Yaskawa INFORM job: KRIS1A.JBI

/JOB
//NAME KRIS1A
//POS
///NPOS 195,195,193,7,0,0
///TOOL 0
///POSTYPE PULSE
///PULSE
C00000=15349,-87390,-111573,-674,86554,-86826
C00001=-110984,-87390,-111570,-673,86559,8331
C00002=-111759,-79535,-69021,-454,64406,8169
C00003=-114095,-78681,-67160,402,63698,7299
C00004=-114095,-78325,-65957,403,63140,7298
C00005=-114095,-78648,-67045,402,63644,7299
C00006=-113114,-93112,-73015,43,59884,7664
C00007=-114174,-91151,-70215,449,59172,7253
C00008=-114269,-89568,-69588,484,59599,7218
C00009=-112804,-96361,-75693,-76,59862,7786
C00010=-111133,-79411,-68712,-683,64284,8404
C00011=-110795,-77497,-66452,-807,63881,8532
C00012=-110795,-77213,-65470,-810,63423,8535
C00013=-111147,-78773,-67027,-680,63577,8402
C00014=-109795,-94038,-73387,-1221,59664,8950
C00015=-110034,-90449,-69592,-1136,59169,8863
C00016=-110197,-88771,-68919,-1070,59614,8797
C00017=-109724,-95740,-76085,-1239,60450,8969
C00018=-97790,-93891,-80845,-5517,64828,13352
C00019=-103428,-49774,-59623,-1029,84980,31565
C00020=-110091,-17957,-40687,2667,97599,44417
C00021=-110679,-18450,-38986,2708,96322,44197
C00022=-110679,-18552,-38259,2706,95822,44188
C00023=-109538,-18108,-38733,2608,96305,44575
C00024=-109458,-19366,-38871,2595,95741,44590
C00025=-109985,-19539,-38909,2643,95690,44414
C00026=-108888,-17833,-38981,2552,96578,44796
C00027=-113591,44136,17002,2949,94129,43179
C00028=-113558,44117,17472,2949,93828,43185
C00029=-113558,44084,18124,2949,93412,43175
C00030=-112698,44382,17754,2873,93761,43471
C00031=-112698,44348,18436,2870,93325,43460
C00032=-113010,44247,18329,2898,93349,43356
C00033=-112698,44452,16728,2876,94428,43485
C00034=-95102,58941,36484,-30043,98742,46310
C00035=-95139,59332,36927,-30037,98667,46316
C00036=-123036,27157,-10763,-19283,86742,21526
C00037=-150798,39984,8064,-10438,77055,13413
C00038=-150701,50951,18953,-20501,80603,7648
C00039=-146523,55066,28554,-32677,81611,-991
C00040=-149211,60857,35994,-32225,79233,-1370
C00041=-149211,60937,37447,-32305,78504,-1162
C00042=-149211,60857,35994,-32225,79233,-1370
C00043=-148938,63495,39015,-32331,78908,-1167
C00044=-149211,60857,35994,-32225,79233,-1370
C00045=-141139,35393,-539,-16647,85388,2500
C00046=-139001,60609,30102,-17411,80166,3961
C00047=-135441,52818,21854,-13680,80270,7361
C00048=-135777,54342,23766,-13597,79830,7293
C00049=-135777,54229,24881,-13624,79108,7374
C00050=-135777,54342,23766,-13597,79830,7293
C00051=-135623,56980,26711,-13659,79411,7392
C00052=-135777,54342,23766,-13597,79830,7293
C00053=-130150,67910,41047,-22097,81612,18545
C00054=-130308,68928,40049,-22014,82627,18301
C00055=-129747,65534,38183,-22158,82221,18578
C00056=-132405,65002,37751,-21584,81519,17750
C00057=-140354,55773,27245,-19636,81172,14970
C00058=-143966,58727,36324,-37580,82061,-623
C00059=-143233,57260,38729,-44506,80254,-83
C00060=-133755,47291,19718,-43086,89514,541
C00061=-130254,27624,-12420,-14523,95031,2735
C00062=-129705,29711,-12872,-15389,97022,78903
C00063=-131005,-814,-31676,-13890,80611,84029
C00064=-141281,-13707,-38556,3093,70993,82901
C00065=-136152,50678,21465,2134,66956,84718
C00066=-128094,56541,22144,-15053,77570,85372
C00067=-123724,-37006,-66316,-16306,84508,85949
C00068=-117270,-70326,-76879,-25476,75485,88799
C00069=-117396,-67861,-71382,-25671,73529,89185
C00070=-117796,-48019,-60604,-25175,76642,88348
C00071=-117668,-98678,-84753,-25780,65584,89666
C00072=-118323,-67765,-71239,-24397,72273,87906
C00073=-118030,-36635,-53581,-24971,77958,87975
C00074=-118346,-17679,-40448,-24750,79381,87560
C00075=-118238,-16726,-43675,-24636,81672,87118
C00076=-116459,-97013,-88147,-26591,69614,90459
C00077=-118030,-36635,-53581,-24971,77958,87975
C00078=-118346,-17679,-40448,-24750,79381,87560
C00079=-118238,-16726,-43675,-24636,81672,87118
C00080=-116459,-97013,-88147,-26591,69614,90459
C00081=-117668,-98678,-84753,-25780,65584,89666
C00082=-118323,-67765,-71239,-24397,72273,87906
C00083=-117271,-70296,-76864,-25474,75490,88797
C00084=-117270,-70326,-76879,-25476,75485,88799
C00085=-117396,-67861,-71382,-25671,73529,89185
C00086=-117796,-48019,-60604,-25175,76642,88348
C00087=-116979,-69120,-74771,-25636,74961,89025
C00088=-117994,-43372,-61454,-24127,91092,85341
C00089=-149498,-32155,-54450,-17063,84771,75512
C00090=-141330,-38704,-51094,-33432,76685,78426
C00091=-130528,-69811,-74379,-36386,79670,81887
C00092=-132947,-100822,-92962,-36380,74991,82451
C00093=15349,-87390,-111573,-674,86554,-86826
C00094=15349,-87390,-111573,-674,86554,-86826
C00095=15349,-87390,-111570,-674,86556,-86825
C00096=3643,-76224,-106676,19950,71810,76872
C00097=15349,-87390,-111570,-674,86556,-86825
C00098=-68824,-87390,-111568,-659,86557,2288
C00099=-102324,-63179,-76492,-4543,93838,9300
C00100=-99268,-62121,-71685,-4896,91607,10397
C00101=-101449,-61888,-70084,-4627,90618,9708
C00102=-101449,-61917,-69079,-4627,89987,9729
C00103=-101449,-61887,-70112,-4627,90636,9704
C00104=-98771,-79826,-78849,-4944,86964,10742
C00105=-97205,-87840,-78173,-7148,76765,11690
C00106=-97422,-86698,-77695,-7095,77039,11596
C00107=-98458,-92698,-83162,-6885,77230,11227
C00108=-70334,-47845,-62333,-11740,90555,19804
C00109=-68889,-44293,-58067,-11955,89977,20346
C00110=-68889,-44364,-57255,-11953,89453,20397
C00111=-68889,-44289,-58112,-11958,90008,20343
C00112=-63676,-56068,-65467,-12713,89294,22180
C00113=-64287,-54843,-62333,-12625,87932,22111
C00114=-64982,-53370,-61506,-12527,88068,21862
C00115=-63556,-56320,-65366,-12731,89128,22240
C00116=-105066,-71099,-78115,-5454,84680,8612
C00117=-111759,-50737,-67326,-4071,88105,-39576
C00118=-98977,-49335,-63615,-15063,89376,-36463
C00119=-99018,-49671,-62454,-15054,88511,-36372
C00120=-99018,-49749,-61553,-15054,87936,-36300
C00121=-99018,-49696,-62187,-15054,88340,-36350
C00122=-100915,-50718,-62779,-14728,87845,-36938
C00123=-100789,-50793,-62111,-14749,87431,-36845
C00124=-100259,-50517,-61951,-14840,87569,-36680
C00125=-101317,-50964,-63445,-14655,88049,-37098
C00126=-98850,-47982,-62812,-15085,89595,-36444
C00127=-99170,-48330,-61581,-15027,88634,-36434
C00128=-99170,-48394,-60912,-15027,88207,-36380
C00129=-99183,-48208,-61790,-15025,88819,-36461
C00130=-101244,-49312,-62437,-14669,88288,-37099
C00131=-100997,-49277,-61381,-14712,87718,-36948
C00132=-100426,-49069,-61280,-14811,87864,-36771
C00133=-101005,-49253,-62663,-14710,88495,-37043
C00134=-99461,-60085,-69932,-19764,73355,-34813
C00135=-111458,-11031,-30949,20838,73112,-726
C00136=-111844,18040,-3295,21202,74863,-1057
C00137=-111040,19701,-1743,20952,74565,-817
C00138=-111040,19683,-1004,20994,74127,-894
C00139=-110997,19721,-1737,20937,74560,-802
C00140=-111040,21506,-67,20957,74469,-835
C00141=-110997,19721,-1737,20937,74560,-802
C00142=-112260,2825,-16849,21290,75457,-1102
C00143=-114727,-25650,-50489,21683,81747,-843
C00144=-114727,-25650,-50489,21683,81747,-843
C00145=-78893,324,-30560,8500,76378,10543
C00146=-78852,391,-30517,8483,76382,10557
C00147=-79073,11131,-13779,8761,71676,10146
C00148=-79035,11094,-12929,8771,71138,10119
C00149=-79073,11131,-13779,8761,71676,10146
C00150=-79422,12797,-12298,8905,71656,10024
C00151=-79073,11131,-13779,8761,71676,10146
C00152=-90006,37360,13465,10198,74665,-440
C00153=-98018,29482,5428,6676,74813,1335
C00154=-100387,34080,10935,-7216,71995,-1662
C00155=-101325,39705,22013,-25009,65580,-3161
C00156=-101232,47576,34073,-36115,63714,-3272
C00157=-99101,24615,5399,-28066,67939,-3113
C00158=-101092,-2809,-21504,5594,61806,151
C00159=-116279,-103565,-87668,15153,52841,-6820
C00160=-136626,-108292,-100051,23905,62636,71559
C00161=-126647,-9226,-38971,10424,73423,75937
C00162=-126713,-9857,-28436,10885,66731,75311
C00163=-125013,58541,36859,10521,61560,75459
C00164=-125013,58363,29682,10151,65819,75847
C00165=-150812,-11611,-31149,38982,76943,71088
C00166=-150812,-11611,-31149,38982,76943,71088
C00167=-179059,-124163,-86099,46721,72567,55901
C00168=-188308,-108023,-75488,46296,78544,54278
C00169=-175675,-91816,-69705,45351,75449,58945
C00170=-166987,-75634,-62751,43730,73998,62467
C00171=-158229,-51102,-50131,41259,73376,66301
C00172=-153526,-28687,-35659,40655,73501,68565
C00173=-150180,-12513,-24053,39553,72873,69823
C00174=-150180,-12464,-30917,38869,76208,71082
C00175=-153640,-28797,-40554,40201,75834,69434
C00176=-153526,-28687,-35659,40655,73501,68565
C00177=-150180,-12513,-24053,39553,72873,69823
C00178=-153459,-29015,-37831,40437,74369,68941
C00179=-158928,-63138,-59452,42454,73735,66180
C00180=-166987,-75634,-62751,43730,73998,62467
C00181=-158229,-51102,-50131,41259,73376,66301
C00182=-167024,-76273,-64991,43548,74788,62799
C00183=-185238,-109581,-79609,46117,78191,55596
C00184=-188308,-108023,-75488,46296,78544,54278
C00185=-175675,-91816,-69705,45351,75449,58945
C00186=-181552,-118218,-82845,46514,74578,55658
C00187=-187474,-110161,-80368,46081,79459,55112
C00188=-145536,-97007,-88996,9555,84002,75248
C00189=-145251,-96121,-85437,9544,82257,75216
C00190=-99167,-97649,-86024,2499,78276,90872
C00191=-118631,-91766,-78858,25217,81137,84835
C00192=-117699,-93504,-86004,20553,84337,85672
C00193=-134531,-91540,-85241,22037,89209,80450
C00194=3161,-91504,-85468,2682,88050,79011
BC00000=115,663699,1075117
BC00001=171753,674879,306456
BC00002=55475,735323,199167
BC00003=55475,735323,199167
BC00004=55475,735323,199167
BC00005=55475,735323,199167
BC00006=55475,735323,199167
BC00007=55475,735323,199167
BC00008=55475,735323,199167
BC00009=55475,735323,199167
BC00010=108320,735323,199167
BC00011=108320,735323,199167
BC00012=108320,735323,199167
BC00013=108320,735323,199167
BC00014=108320,735323,199167
BC00015=108320,735323,199167
BC00016=108320,735323,199167
BC00017=108320,735323,199167
BC00018=108320,735323,199167
BC00019=108320,735323,199167
BC00020=108320,735323,199167
BC00021=108320,735323,199167
BC00022=108320,735323,199167
BC00023=108320,735323,199167
BC00024=108320,735323,199167
BC00025=108320,735323,199167
BC00026=108320,735323,199167
BC00027=108320,749563,199167
BC00028=108320,749563,199167
BC00029=108320,749563,199167
BC00030=108320,749563,199167
BC00031=108320,749563,199167
BC00032=108320,749563,199166
BC00033=108320,749563,199167
BC00034=108320,749563,199167
BC00035=108320,749563,199167
BC00036=153902,806828,124230
BC00037=190527,806828,124230
BC00038=190527,806828,124230
BC00039=190527,806828,124230
BC00040=190526,806828,124220
BC00041=190526,806828,124220
BC00042=190526,806828,124220
BC00043=190526,806828,124220
BC00044=190526,806828,124220
BC00045=190527,806828,124230
BC00046=190527,806828,124230
BC00047=170092,806828,124230
BC00048=170092,806828,124230
BC00049=170092,806828,124230
BC00050=170092,806828,124230
BC00051=170092,806828,124230
BC00052=170092,806828,124230
BC00053=170093,806828,124227
BC00054=170093,806828,124227
BC00055=170093,806828,124227
BC00056=170093,806828,124224
BC00057=170093,806828,124224
BC00058=170093,806828,124224
BC00059=170093,806828,124227
BC00060=170093,806828,124227
BC00061=170093,806828,124227
BC00062=170093,806828,124227
BC00063=170093,806828,124227
BC00064=170093,806828,124227
BC00065=170093,806828,124227
BC00066=170093,806828,124227
BC00067=170093,806828,124227
BC00068=170093,743154,124227
BC00069=170093,743154,124227
BC00070=170093,743154,124227
BC00071=170093,806828,124227
BC00072=170093,806828,124227
BC00073=170093,806828,124227
BC00074=170093,806828,124227
BC00075=170093,806828,124227
BC00076=170093,806828,124227
BC00077=170093,806828,124227
BC00078=170093,806828,124227
BC00079=170093,806828,124227
BC00080=170093,806828,124227
BC00081=170093,806828,124227
BC00082=170093,806828,124227
BC00083=170093,806828,124227
BC00084=170093,743154,124227
BC00085=170093,743154,124227
BC00086=170093,743154,124227
BC00087=170093,743154,124227
BC00088=170093,743154,124227
BC00089=170093,743154,124227
BC00090=170093,743154,124227
BC00091=170093,743154,124227
BC00092=170093,743154,124227
BC00093=115,663699,1075117
BC00094=115,663699,1075117
BC00095=115,663700,1075116
BC00096=199464,674570,1075173
BC00097=141263,687330,337717
BC00098=222435,751088,164876
BC00099=279925,751088,164876
BC00100=279925,751088,164876
BC00101=279925,751088,164876
BC00102=279925,751088,164876
BC00103=279925,751088,164876
BC00104=279925,751088,164876
BC00105=279925,751088,164876
BC00106=279925,751088,164876
BC00107=279925,751088,164876
BC00108=279925,751088,164876
BC00109=279925,751088,164876
BC00110=279925,751088,164876
BC00111=279925,751088,164876
BC00112=279925,751088,164876
BC00113=279925,751088,164876
BC00114=279925,751088,164876
BC00115=279925,751088,164876
BC00116=279925,751088,164876
BC00117=279925,751088,164876
BC00118=279925,751088,164876
BC00119=279925,751088,164876
BC00120=279925,751088,164876
BC00121=279925,751088,164876
BC00122=279925,751088,164876
BC00123=279925,751088,164876
BC00124=279925,751088,164876
BC00125=279925,751088,164876
BC00126=279925,839714,164876
BC00127=279925,839714,164876
BC00128=279925,839714,164876
BC00129=279925,839714,164876
BC00130=279925,839714,164876
BC00131=279925,839714,164876
BC00132=279925,839714,164876
BC00133=279925,839714,164876
BC00134=279925,839714,164876
BC00135=279925,839714,164876
BC00136=279925,834738,164876
BC00137=279925,834738,164876
BC00138=279925,834738,164876
BC00139=279925,834738,164876
BC00140=279925,834738,164876
BC00141=279925,834738,164876
BC00142=279925,834738,164876
BC00143=279925,834738,164876
BC00144=279925,762190,164876
BC00145=244896,762190,164876
BC00146=278481,826600,138122
BC00147=278481,826600,138122
BC00148=278481,826600,138122
BC00149=278481,826600,138122
BC00150=278481,826600,138122
BC00151=278481,826600,138122
BC00152=302666,794256,164873
BC00153=326440,794256,164873
BC00154=326440,794256,164873
BC00155=326440,794254,164874
BC00156=326440,794256,164873
BC00157=326440,794256,164873
BC00158=326440,794256,164873
BC00159=326440,794256,164873
BC00160=326440,794256,164873
BC00161=326440,794256,164873
BC00162=326885,794948,164297
BC00163=326885,794948,164297
BC00164=326885,794948,164297
BC00165=326885,794948,164297
BC00166=326885,794948,164297
BC00167=326885,794948,164297
BC00168=326885,794948,164297
BC00169=326885,794948,164297
BC00170=326885,794948,164297
BC00171=326885,794948,164297
BC00172=326885,794948,164297
BC00173=326885,794948,164297
BC00174=326885,794948,164297
BC00175=326885,794948,164297
BC00176=326885,794948,164297
BC00177=326885,794948,164297
BC00178=326885,794948,164297
BC00179=326885,794948,164297
BC00180=326885,794948,164297
BC00181=326885,794948,164297
BC00182=326885,794948,164297
BC00183=326885,794948,164297
BC00184=326885,794948,164297
BC00185=326885,794948,164297
BC00186=326885,794948,164297
BC00187=326885,794948,164297
BC00188=326885,794948,164297
BC00189=326885,794948,164297
BC00190=326885,794948,164297
BC00191=326885,794948,164295
BC00192=326885,794948,164295
BC00193=326885,737668,213736
BC00194=87842,675035,1040975
EC00000=798157,0
EC00001=798154,2
EC00002=798154,2
EC00003=798154,2
EC00004=798154,2
EC00005=798154,2
EC00006=798154,2
EC00007=798154,2
EC00008=798154,2
EC00009=798154,2
EC00010=798154,2
EC00011=798154,2
EC00012=798154,2
EC00013=798154,2
EC00014=798154,2
EC00015=798154,2
EC00016=798154,2
EC00017=798154,2
EC00018=798154,2
EC00019=798154,2
EC00020=798154,2
EC00021=798154,2
EC00022=798154,2
EC00023=798154,2
EC00024=798154,2
EC00025=798154,2
EC00026=798154,2
EC00027=798154,2
EC00028=798154,2
EC00029=798154,2
EC00030=798154,2
EC00031=798154,2
EC00032=798153,2
EC00033=798154,2
EC00034=798154,2
EC00035=798154,2
EC00036=798154,2
EC00037=798154,2
EC00038=798154,2
EC00039=798154,2
EC00040=798150,3
EC00041=798150,3
EC00042=798150,3
EC00043=798150,3
EC00044=798150,3
EC00045=798154,2
EC00046=798154,2
EC00047=798154,2
EC00048=798154,2
EC00049=798154,2
EC00050=798154,2
EC00051=798154,2
EC00052=798154,2
EC00053=798153,2
EC00054=798151,3
EC00055=798151,3
EC00056=798152,2
EC00057=798153,2
EC00058=798153,2
EC00059=798153,2
EC00060=798153,2
EC00061=798153,2
EC00062=798153,2
EC00063=798153,2
EC00064=798153,2
EC00065=798153,2
EC00066=798153,2
EC00067=798153,2
EC00068=798153,2
EC00069=798153,2
EC00070=798153,2
EC00071=798153,2
EC00072=798153,2
EC00073=798153,2
EC00074=798153,2
EC00075=798153,2
EC00076=798153,2
EC00077=798153,2
EC00078=798153,2
EC00079=798153,2
EC00080=798153,2
EC00081=798153,2
EC00082=798153,2
EC00083=798153,2
EC00084=798153,2
EC00085=798153,2
EC00086=798153,2
EC00087=798153,2
EC00088=798153,2
EC00089=798153,2
EC00090=798153,2
EC00091=798157,0
EC00092=93266,10480
EC00093=184298,1105644
EC00094=798157,1112952
EC00095=798157,1112952
EC00096=798156,1112951
EC00097=798156,1112951
EC00098=798156,1112951
EC00099=798156,1112951
EC00100=798156,1112951
EC00101=798156,1112951
EC00102=798156,1112951
EC00103=798156,1112951
EC00104=798156,1112951
EC00105=798156,1112951
EC00106=798156,1112951
EC00107=798156,1112951
EC00108=798156,1112951
EC00109=798156,1112951
EC00110=798156,1112951
EC00111=798156,1112951
EC00112=798156,1112951
EC00113=798156,1112951
EC00114=798156,1112951
EC00115=798156,1112951
EC00116=798156,1112951
EC00117=798156,1112951
EC00118=798156,1112951
EC00119=798156,1112951
EC00120=798156,1112951
EC00121=798156,1112951
EC00122=798156,1112951
EC00123=798156,1112951
EC00124=798156,1112951
EC00125=798156,1112951
EC00126=798156,1112951
EC00127=798156,1112951
EC00128=798156,1112951
EC00129=798156,1112951
EC00130=798156,1112951
EC00131=798156,1112951
EC00132=798156,1112951
EC00133=798156,1112951
EC00134=798156,1112951
EC00135=798156,1112951
EC00136=798156,1112951
EC00137=798156,1112951
EC00138=798156,1112951
EC00139=798156,1112951
EC00140=798156,1112951
EC00141=798156,1112951
EC00142=798156,1112951
EC00143=798156,1112951
EC00144=798156,1112951
EC00145=798156,1112951
EC00146=798156,1112951
EC00147=798156,1112951
EC00148=798156,1112951
EC00149=798156,1112951
EC00150=798155,1112950
EC00151=798155,1112950
EC00152=798155,1112950
EC00153=798155,1112950
EC00154=798155,1112950
EC00155=798155,1112950
EC00156=798155,1112950
EC00157=798155,1112950
EC00158=798155,1112950
EC00159=798155,1112950
EC00160=798155,1112950
EC00161=798155,1112950
EC00162=798155,1112950
EC00163=798155,1112950
EC00164=798155,1112950
EC00165=798155,1112950
EC00166=798155,1112950
EC00167=798155,1112950
EC00168=798155,1112950
EC00169=798155,1112950
EC00170=798155,1112950
EC00171=798155,1112950
EC00172=798155,1112950
EC00173=798155,1112950
EC00174=798155,1112950
EC00175=798155,1112950
EC00176=798155,1112950
EC00177=798155,1112950
EC00178=798155,1112950
EC00179=798155,1112950
EC00180=798155,1112950
EC00181=798155,1112950
EC00182=798155,1112950
EC00183=798155,1112950
EC00184=798155,1112950
EC00185=798155,1112950
EC00186=798155,1112950
EC00187=798155,1112950
EC00188=798155,1112950
EC00189=798154,1112948
EC00190=798154,1112948
EC00191=798154,1112948
EC00192=798154,1103372
///POSTYPE BASE
///RECTAN
///RCONF 0,0,0,0,0,0,0,0,0,0,0,0,0,0,0,0,0,0,0,0,0,0,0,0
P00006=0.222,-3.123,-1.508,0.0000,0.0000,0.0000
P00021=-0.225,-6.128,-0.405,0.0000,0.0000,0.0000
P00022=0.222,-3.123,-1.508,0.0000,0.0000,0.0000
P00023=0.143,-0.036,0.682,0.0000,0.0000,0.0000
P00024=0.145,-0.552,1.326,0.0000,0.0000,0.0000
P00025=-2.003,0.006,0.728,0.0000,0.0000,0.0000
P00026=0.562,-0.002,-0.337,0.0000,0.0000,0.0000
//INST
///DATE 2025/03/14 13:10
///ATTR SC,RW
///GROUP1 RB1,BS1
///GROUP2 ST1
NOP
CALL JOB:CLEAN-R1_KM_3P
MOVJ C00000 BC00000 VJ=100.00  +MOVJ EC00000 VJ=100.00
MOVJ C00001 BC00001 VJ=100.00  +MOVJ EC00001 VJ=100.00
MOVJ C00002 BC00002 VJ=100.00  +MOVJ EC00002 VJ=100.00
SMOVL C00003 BC00003 V=100.0  +MOVJ EC00003
SREFP 3 C00004 BC00004  +REFP EC00004
CALL JOB:SEARCH-R1-S13D
SET P023 P006
SFTON3D P023
SMOVL C00005 BC00005 V=133.3  +MOVJ EC00005
SMOVL C00006 BC00006 V=133.3  +MOVJ EC00006
SMOVL C00007 BC00007 V=133.3  +MOVJ EC00007
SREFP 3 C00008 BC00008  +REFP EC00008
CALL JOB:SEARCH-R1-S13D
SET P023 P006
SFTON3D P023
SMOVL C00009 BC00009 V=166.7  +MOVJ EC00009
SFTOF3D
SMOVL C00010 BC00010 V=250.0  +MOVJ EC00010
SMOVL C00011 BC00011 V=100.0  +MOVJ EC00011
SREFP 3 C00012 BC00012  +REFP EC00012
CALL JOB:SEARCH-R1-S13D
SET P024 P006
SFTON3D P024
SMOVL C00013 BC00013 V=133.3  +MOVJ EC00013
SMOVL C00014 BC00014 V=133.3  +MOVJ EC00014
SMOVL C00015 BC00015 V=133.3  +MOVJ EC00015
SREFP 3 C00016 BC00016  +REFP EC00016
CALL JOB:SEARCH-R1-S13D
SET P024 P006
SFTON3D P024
SMOVL C00017 BC00017 V=166.7  +MOVJ EC00017
SFTOF3D
MOVJ C00018 BC00018 VJ=100.00  +MOVJ EC00018 VJ=100.00
MOVJ C00019 BC00019 VJ=100.00  +MOVJ EC00019 VJ=100.00
MOVJ C00020 BC00020 VJ=100.00  +MOVJ EC00020 VJ=100.00
SMOVL C00021 BC00021 V=100.0  +MOVJ EC00021
SREFP 3 C00022 BC00022  +REFP EC00022
CALL JOB:SEARCH-R1-S13D
SET P025 P006
SFTON3D P025
SMOVL C00023 BC00023 V=100.0  +MOVJ EC00023
SMOVL C00024 BC00024 V=100.0  +MOVJ EC00024
SREFP 3 C00025 BC00025  +REFP EC00025
CALL JOB:SEARCH-R1-S13D
SET P025 P006
SFTON3D P025
SMOVL C00026 BC00026 V=100.0  +MOVJ EC00026
SFTOF3D
SMOVL C00027 BC00027 V=500.0  +MOVJ EC00027
SMOVL C00028 BC00028 V=100.0  +MOVJ EC00028
SREFP 3 C00029 BC00029  +REFP EC00029
CALL JOB:SEARCH-R1-S13D
SET P026 P006
SFTON3D P026
SMOVL C00030 BC00030 V=133.3  +MOVJ EC00030
SMOVL C00031 BC00031 V=100.0  +MOVJ EC00031
SREFP 3 C00032 BC00032  +REFP EC00032
CALL JOB:SEARCH-R1-S13D
SET P026 P006
SFTON3D P026
SMOVL C00033 BC00033 V=166.7  +MOVJ EC00033
SFTOF3D
SMOVL C00034 BC00034 V=500.0  +MOVJ EC00034
MOVJ C00035 BC00035 VJ=100.00  +MOVJ EC00035 VJ=100.00
MOVJ C00036 BC00036 VJ=100.00  +MOVJ EC00036 VJ=20.00
MOVJ C00037 BC00037 VJ=20.00  +MOVJ EC00037 VJ=20.00
MOVJ C00038 BC00038 VJ=20.00  +MOVJ EC00038 VJ=20.00
MOVJ C00039 BC00039 VJ=20.00  +MOVJ EC00039 VJ=20.00
SMOVL C00040 BC00040 V=100.0  +MOVJ EC00040
SREFP 3 C00041 BC00041  +REFP EC00041
CALL JOB:SEARCH-R1-S13D
SET P022 P006
SFTON3D P022
SMOVL C00042 BC00042 V=100.0  +MOVJ EC00042
SREFP 3 C00043 BC00043  +REFP EC00043
CALL JOB:SEARCH-R1-S13D
SET P022 P006
SFTON3D P022
SMOVL C00044 BC00044 V=100.0  +MOVJ EC00044
SFTOF3D
MOVL C00045 BC00045 V=500.0  +MOVJ EC00045 VJ=20.00
MOVL C00046 BC00046 V=500.0  +MOVJ EC00046 VJ=20.00
SMOVL C00047 BC00047 V=500.0  +MOVJ EC00047
SMOVL C00048 BC00048 V=100.0  +MOVJ EC00048
SREFP 3 C00049 BC00049  +REFP EC00049
CALL JOB:SEARCH-R1-S13D
SET P021 P006
SFTON3D P021
SMOVL C00050 BC00050 V=100.0  +MOVJ EC00050
SREFP 3 C00051 BC00051  +REFP EC00051
CALL JOB:SEARCH-R1-S13D
SET P021 P006
SFTON3D P021
SMOVL C00052 BC00052 V=100.0  +MOVJ EC00052
MACRO1 MJ#(0) ARGF21
SMOVL C00053 BC00053 V=250.0  +MOVJ EC00053
REFP 1 RB1 C00054 BC00054
REFP 2 RB1 C00055 BC00055
ARCON
SWVON WEV#(100)
SMOVL C00056 BC00056 V=8.3  +MOVJ EC00054
SFTON3D P022
SMOVL C00057 BC00057 V=8.3  +MOVJ EC00055
SMOVL C00058 BC00058 V=8.3  +MOVJ EC00056
SMOVL C00059 BC00059 V=8.3  +MOVJ EC00057
ARCOF
SWVOF
SFTOF3D
SMOVL C00060 BC00060 V=333.3  +MOVJ EC00058
SMOVL C00061 BC00061 V=666.7  +MOVJ EC00059
MOVJ C00062 BC00062 VJ=100.00  +MOVJ EC00060 VJ=20.00
MOVJ C00063 BC00063 VJ=70.00  +MOVJ EC00061 VJ=20.00
MACRO1 MJ#(0) ARGF20
SFTON3D P025
SMOVL C00064 BC00064 V=250.0  +MOVJ EC00062
ARCON
SFTON3D P026
SMOVL C00065 BC00065 V=7.5  +MOVJ EC00063
ARCOF
SWVOF
SFTOF3D
SMOVL C00066 BC00066 V=333.3  +MOVJ EC00064
SMOVL C00067 BC00067 V=666.7  +MOVJ EC00065
SFTOF3D
MACRO1 MJ#(0) ARGF14
SMOVL C00068 BC00068 V=500.0  +MOVJ EC00066
SFTON3D P025
SMOVL C00069 BC00069 V=166.7  +MOVJ EC00067
ARCON
SWVON WEV#(20)
SMOVL C00070 BC00070 V=10.0  +MOVJ EC00068
SFTON3D P025
SMOVL C00071 BC00071 V=10.0  +MOVJ EC00069
SFTON3D P026
SMOVL C00072 BC00072 V=10.0  +MOVJ EC00070
SFTON3D P026
SMOVL C00073 BC00073 V=10.0  +MOVJ EC00071
SMOVL C00074 BC00074 V=10.0  +MOVJ EC00072
ARCOF
SWVOF
SMOVL C00075 BC00075 V=250.0  +MOVJ EC00073
SMOVL C00076 BC00076 V=500.0  +MOVJ EC00074
COMM MACRO1 MJ#(0) ARGF14
COMM SFTON3D P026
COMM SMOVL C00077 BC00077 V=250.0  +MOVJ EC00075
COMM ARCON
COMM SWVON WEV#(20)
COMM SMOVL C00078 BC00078 V=10.0  +MOVJ EC00076
COMM ARCOF
COMM SWVOF
COMM SMOVL C00079 BC00079 V=250.0  +MOVJ EC00077
COMM SMOVL C00080 BC00080 V=500.0  +MOVJ EC00078
COMM SFTON3D P025
COMM SMOVL C00081 BC00081 V=166.7  +MOVJ EC00079
COMM ARCON
COMM SWVON WEV#(20)
COMM SFTON3D P026
COMM SMOVL C00082 BC00082 V=9.2  +MOVJ EC00080
COMM ARCOF
COMM SWVOF
COMM SMOVL C00083 BC00083 V=250.0  +MOVJ EC00081
COMM SFTOF3D
COMM SMOVL C00084 BC00084 V=500.0  +MOVJ EC00082
COMM SFTON3D P025
COMM SMOVL C00085 BC00085 V=166.7  +MOVJ EC00083
COMM ARCON
COMM SWVON WEV#(20)
COMM SMOVL C00086 BC00086 V=10.0  +MOVJ EC00084
COMM ARCOF
COMM SWVOF
SFTOF3D
SMOVL C00087 BC00087 V=333.3  +MOVJ EC00085
SFTON3D P024
SMOVL C00088 BC00088 V=166.7  +MOVJ EC00086
ARCON
SWVON WEV#(20)
SFTON3D P023
SMOVL C00089 BC00089 V=12.5  +MOVJ EC00087
SMOVL C00090 BC00090 V=12.5  +MOVJ EC00088
ARCOF
SWVOF
SFTOF3D
SMOVL C00091 BC00091 V=500.0  +MOVJ EC00089
SMOVL C00092 BC00092 V=1000.0  +MOVJ EC00090
MOVJ C00093 BC00093 VJ=100.00  +MOVJ EC00091 VJ=20.00
MOVJ C00094 BC00094 VJ=100.00  +MOVJ EC00092 VJ=100.00
MOVJ C00095 BC00095 VJ=100.00  +MOVJ EC00093 VJ=100.00
MOVJ C00096 BC00096 VJ=100.00  +MOVJ EC00094 VJ=100.00
'DRUGA STRONA
CALL JOB:CLEAN-R1_KM_NEW
MOVJ C00097 BC00097 VJ=100.00  +MOVJ EC00095 VJ=100.00
MOVJ C00098 BC00098 VJ=100.00  +MOVJ EC00096 VJ=100.00
MOVJ C00099 BC00099 VJ=100.00  +MOVJ EC00097 VJ=100.00
MOVJ C00100 BC00100 VJ=100.00  +MOVJ EC00098 VJ=100.00
SMOVL C00101 BC00101 V=166.7  +MOVJ EC00099
SREFP 3 C00102 BC00102  +REFP EC00100
CALL JOB:SEARCH-R1-S13D
SET P023 P006
SFTON3D P023
SMOVL C00103 BC00103 V=250.0  +MOVJ EC00101
SMOVL C00104 BC00104 V=250.0  +MOVJ EC00102
SMOVL C00105 BC00105 V=250.0  +MOVJ EC00103
SREFP 3 C00106 BC00106  +REFP EC00104
CALL JOB:SEARCH-R1-S13D
SET P023 P006
SFTON3D P023
SFTOF3D
SMOVL C00107 BC00107 V=250.0  +MOVJ EC00105
SMOVL C00108 BC00108 V=250.0  +MOVJ EC00106
SMOVL C00109 BC00109 V=250.0  +MOVJ EC00107
SREFP 3 C00110 BC00110  +REFP EC00108
CALL JOB:SEARCH-R1-S13D
SET P024 P006
SFTON3D P024
SMOVL C00111 BC00111 V=250.0  +MOVJ EC00109
SMOVL C00112 BC00112 V=250.0  +MOVJ EC00110
SMOVL C00113 BC00113 V=250.0  +MOVJ EC00111
SREFP 3 C00114 BC00114  +REFP EC00112
CALL JOB:SEARCH-R1-S13D
SET P024 P006
SFTON3D P024
SFTOF3D
SMOVL C00115 BC00115 V=250.0  +MOVJ EC00113
MOVJ C00116 BC00116 VJ=100.00  +MOVJ EC00114 VJ=100.00
MOVJ C00117 BC00117 VJ=100.00  +MOVJ EC00115 VJ=100.00
MOVJ C00118 BC00118 VJ=100.00  +MOVJ EC00116 VJ=100.00
SMOVL C00119 BC00119 V=250.0  +MOVJ EC00117
SREFP 3 C00120 BC00120  +REFP EC00118
CALL JOB:SEARCH-R1-S13D
SET P025 P006
SFTON3D P025
SMOVL C00121 BC00121 V=250.0  +MOVJ EC00119
SMOVL C00122 BC00122 V=250.0  +MOVJ EC00120
SMOVL C00123 BC00123 V=100.0  +MOVJ EC00121
SREFP 3 C00124 BC00124  +REFP EC00122
CALL JOB:SEARCH-R1-S13D
SET P025 P006
SFTON3D P025
SFTOF3D
SMOVL C00125 BC00125 V=100.0  +MOVJ EC00123
SMOVL C00126 BC00126 V=333.3  +MOVJ EC00124
SMOVL C00127 BC00127 V=250.0  +MOVJ EC00125
SREFP 3 C00128 BC00128  +REFP EC00126
CALL JOB:SEARCH-R1-S13D
SET P026 P006
SFTON3D P026
SMOVL C00129 BC00129 V=250.0  +MOVJ EC00127
SMOVL C00130 BC00130 V=250.0  +MOVJ EC00128
SMOVL C00131 BC00131 V=100.0  +MOVJ EC00129
SREFP 3 C00132 BC00132  +REFP EC00130
CALL JOB:SEARCH-R1-S13D
SET P026 P006
SFTON3D P026
SFTOF3D
SMOVL C00133 BC00133 V=250.0  +MOVJ EC00131
SMOVL C00134 BC00134 V=333.3  +MOVJ EC00132
MOVJ C00135 BC00135 VJ=20.00  +MOVJ EC00133 VJ=20.00
MOVJ C00136 BC00136 VJ=20.00  +MOVJ EC00134 VJ=20.00
SMOVL C00137 BC00137 V=250.0  +MOVJ EC00135
SREFP 3 C00138 BC00138  +REFP EC00136
CALL JOB:SEARCH-R1-S13D
SET P021 P006
SFTON3D P021
SMOVL C00139 BC00139 V=250.0  +MOVJ EC00137
SREFP 3 C00140 BC00140  +REFP EC00138
CALL JOB:SEARCH-R1-S13D
SET P021 P006
SFTON3D P021
SFTOF3D
SMOVL C00141 BC00141 V=250.0  +MOVJ EC00139
MOVL C00142 BC00142 V=250.0  +MOVJ EC00140 VJ=20.00
MOVL C00143 BC00143 V=333.3  +MOVJ EC00141 VJ=20.00
SMOVL C00144 BC00144 V=1000.0  +MOVJ EC00142
SMOVL C00145 BC00145 V=1000.0  +MOVJ EC00143
SMOVL C00146 BC00146 V=250.0  +MOVJ EC00144
SMOVL C00147 BC00147 V=250.0  +MOVJ EC00145
SREFP 3 C00148 BC00148  +REFP EC00146
CALL JOB:SEARCH-R1-S13D
SET P022 P006
SFTON3D P022
SMOVL C00149 BC00149 V=250.0  +MOVJ EC00147
SREFP 3 C00150 BC00150  +REFP EC00148
CALL JOB:SEARCH-R1-S13D
SET P022 P006
SFTON3D P022
SFTOF3D
SMOVL C00151 BC00151 V=250.0  +MOVJ EC00149
MACRO1 MJ#(0) ARGF21
SFTON3D P022
SMOVL C00152 BC00152 V=250.0  +MOVJ EC00150
ARCON
SWVON WEV#(100)
SMOVL C00153 BC00153 V=8.3  +MOVJ EC00151
SMOVL C00154 BC00154 V=8.3  +MOVJ EC00152
SMOVL C00155 BC00155 V=8.3  +MOVJ EC00153
SMOVL C00156 BC00156 V=8.3  +MOVJ EC00154
ARCOF
SWVOF
SMOVL C00157 BC00157 V=250.0  +MOVJ EC00155
SMOVL C00158 BC00158 V=500.0  +MOVJ EC00156
MOVJ C00159 BC00159 VJ=50.00  +MOVJ EC00157 VJ=20.00
MOVJ C00160 BC00160 VJ=100.00  +MOVJ EC00158 VJ=20.00
MOVJ C00161 BC00161 VJ=40.00  +MOVJ EC00159 VJ=20.00
MACRO1 MJ#(0) ARGF20
SFTON3D P025
SMOVL C00162 BC00162 V=133.3 PL=0  +MOVJ EC00160
ARCON
SFTON3D P026
SMOVL C00163 BC00163 V=6.7  +MOVJ EC00161
ARCOF
SWVOF
SMOVL C00164 BC00164 V=250.0  +MOVJ EC00162
SFTOF3D
SFTON3D P026
SMOVL C00165 BC00165 V=500.0  +MOVJ EC00163
SFTOF3D
MACRO1 MJ#(0) ARGF14
SMOVL C00166 BC00166 V=500.0  +MOVJ EC00164
SMOVL C00167 BC00167 V=500.0  +MOVJ EC00165
SFTON3D P025
SMOVL C00168 BC00168 V=166.7 PL=0  +MOVJ EC00166
ARCON
SWVON WEV#(20)
SMOVL C00169 BC00169 V=10.0  +MOVJ EC00167
SFTON3D P026
SMOVL C00170 BC00170 V=10.0  +MOVJ EC00168
SMOVL C00171 BC00171 V=10.0  +MOVJ EC00169
SMOVL C00172 BC00172 V=10.0  +MOVJ EC00170
SMOVL C00173 BC00173 V=10.0  +MOVJ EC00171
ARCOF
SWVOF
SFTOF3D
SMOVL C00174 BC00174 V=333.3  +MOVJ EC00172
COMM SMOVL C00175 BC00175 V=250.0  +MOVJ EC00173
COMM SMOVL C00176 BC00176 V=250.0  +MOVJ EC00174
COMM ARCON
COMM SWVON WEV#(20)
COMM SMOVL C00177 BC00177 V=10.0  +MOVJ EC00175
COMM ARCOF
COMM SWVOF
COMM SFTOF3D
COMM SMOVL C00178 BC00178 V=250.0  +MOVJ EC00176
COMM SMOVL C00179 BC00179 V=250.0  +MOVJ EC00177
COMM SFTON3D P026
COMM SMOVL C00180 BC00180 V=250.0  +MOVJ EC00178
COMM ARCON
COMM SWVON WEV#(20)
COMM SMOVL C00181 BC00181 V=10.0  +MOVJ EC00179
COMM ARCOF
COMM SWVOF
COMM SMOVL C00182 BC00182 V=250.0  +MOVJ EC00180
COMM SMOVL C00183 BC00183 V=250.0  +MOVJ EC00181
COMM SFTOF3D
COMM SFTON3D P025
COMM SMOVL C00184 BC00184 V=250.0  +MOVJ EC00182
COMM ARCON
COMM SWVON WEV#(20)
COMM SMOVL C00185 BC00185 V=10.0  +MOVJ EC00183
COMM ARCOF
COMM SWVOF
SMOVL C00186 BC00186 V=500.0  +MOVJ EC00184
SMOVL C00187 BC00187 V=250.0  +MOVJ EC00185
MOVL C00188 BC00188 V=250.0  +MOVJ EC00186 VJ=100.00
SFTON3D P023
SMOVL C00189 BC00189 V=250.0  +MOVJ EC00187
ARCON
SWVON WEV#(20)
SFTON3D P024
SMOVL C00190 BC00190 V=11.7  +MOVJ EC00188
SMOVL C00191 BC00191 V=11.7  +MOVJ EC00189
ARCOF
SWVOF
SFTOF3D
SMOVL C00192 BC00192 V=250.0  +MOVJ EC00190
MOVJ C00193 BC00193 VJ=100.00  +MOVJ EC00191 VJ=20.00
MOVJ C00194 BC00194 VJ=100.00  +MOVJ EC00192 VJ=100.00
END
